// TIA Portal V16 export
// export: Created 2022-01-20T18:36:27.7444699Z, ExportSetting WithDefaults, DisplayName Totally Integrated Automation Portal, DisplayVersion V16, DisplayName TIA Portal Version Control Interface, DisplayVersion V16, DisplayName TIA Portal Openness, DisplayVersion V16, DisplayName STEP 7 Professional, DisplayVersion V16, DisplayName STEP 7 Safety, DisplayVersion V16, DisplayName WinCC Advanced, DisplayVersion V16
FUNCTION_BLOCK "TCPIP_COMMS"   // FB1, LAD
{ S7_Optimized_Access := 'TRUE' }
VERSION : 0.1
// stored: AutoNumber true, IsIECCheckEnabled false, IsRetainMemResEnabled false, MemoryReserve 100, SetENOAutomatically false, UDAEnableTagReadback false
   VAR
      TCON : Struct
         REQ : Bool;
         DONE : Bool;
         BUSY : Bool;
         ERROR : Bool;
         STATUS : UInt;
         DONESAVE : Bool;
      END_STRUCT;
      TDISCON : Struct
         REQ : Bool;
         DONE : Bool;
         BUSY : Bool;
         ERROR : Bool;
         DONESAVE : Bool;
         STATUS : UInt;
      END_STRUCT;
      TSEND : Struct
         REQ : Bool;
         DONE : Bool;
         BUSY : Bool;
         ERROR : Bool;
         DONESAVE : Bool;
         STATUS : UInt;
      END_STRUCT;
      TRCV : Struct
         EN_R : Bool;
         NDR : Bool;
         BUSY : Bool;
         ERROR : Bool;
         STATUS : UInt;
         RCVD_LEN : UDInt;
      END_STRUCT;
      ReceivedString : String;
      TCON_DB { ExternalAccessible := 'False'; ExternalVisible := 'False'; ExternalWritable := 'False'} : TCON;
      TDISCON_DB { ExternalAccessible := 'False'; ExternalVisible := 'False'; ExternalWritable := 'False'} : TDISCON;
      TSEND_DB { ExternalAccessible := 'False'; ExternalVisible := 'False'; ExternalWritable := 'False'} : TSEND;
      TRCV_DB { ExternalAccessible := 'False'; ExternalVisible := 'False'; ExternalWritable := 'False'} : TRCV;
   END_VAR
BEGIN

REGION Network 1: TCON
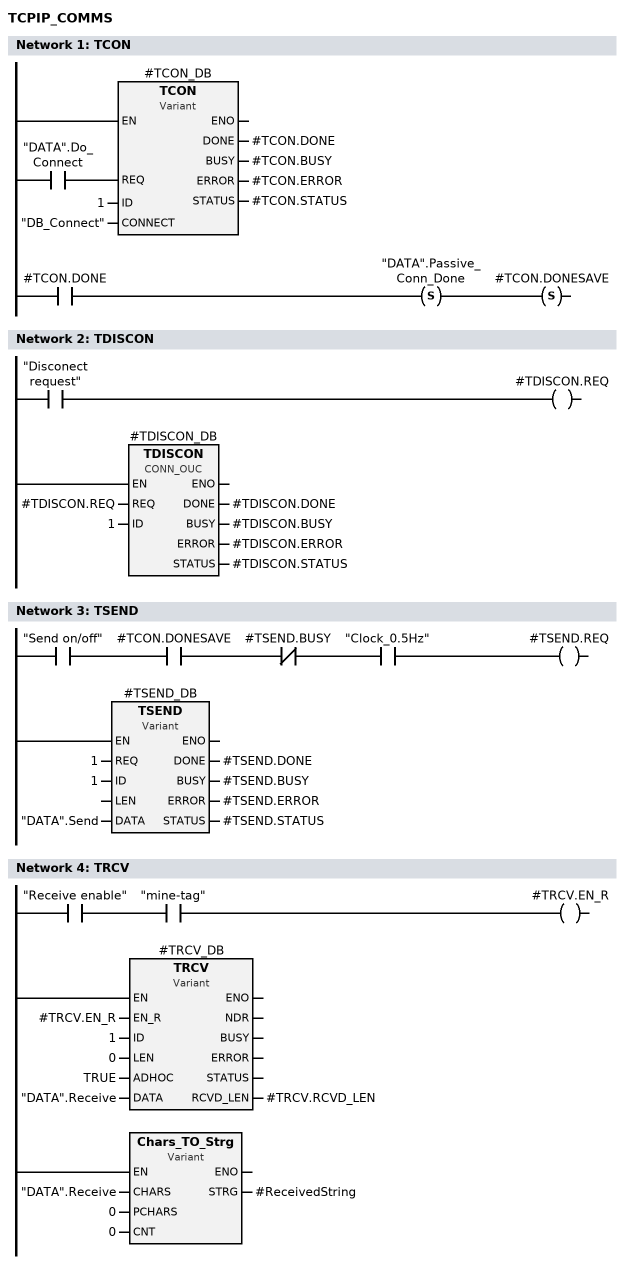
   RUNG wire#powerrail
      { S7_Templates := "[con_type := Variant, id_type := CONN_OUC]" } #TCON_DB.TCON(REQ := wire#w1, ID := 1, CONNECT := "DB_Connect", DONE => #TCON.DONE, BUSY => #TCON.BUSY, ERROR => #TCON.ERROR, STATUS => #TCON.STATUS)
   END_RUNG
   RUNG wire#powerrail
      Contact( "DATA".Do_Connect )
   END_RUNG wire#w1
   RUNG wire#powerrail
      Contact( #TCON.DONE )
      S_Coil( "DATA".Passive_Conn_Done )
      S_Coil( #TCON.DONESAVE )
   END_RUNG
   // the same network as SCL:
   #TCON_DB(REQ := "DATA".Do_Connect,   // TCON
            ID := 1,
            CONNECT := "DB_Connect",
            DONE => #TCON.DONE,
            BUSY => #TCON.BUSY,
            ERROR => #TCON.ERROR,
            STATUS => #TCON.STATUS);
   IF #TCON.DONE THEN
       "DATA".Passive_Conn_Done := TRUE;
       #TCON.DONESAVE := TRUE;
   END_IF;
END_REGION

REGION Network 2: TDISCON
   RUNG wire#powerrail
      Contact( "Disconect request" )
      Coil( #TDISCON.REQ )
   END_RUNG
   RUNG wire#powerrail
      { S7_Templates := "id_type := CONN_OUC" } #TDISCON_DB.TDISCON(REQ := #TDISCON.REQ, ID := 1, DONE => #TDISCON.DONE, BUSY => #TDISCON.BUSY, ERROR => #TDISCON.ERROR, STATUS => #TDISCON.STATUS)
   END_RUNG
   // the same network as SCL:
   #TDISCON.REQ := "Disconect request";
   #TDISCON_DB(REQ := #TDISCON.REQ,   // TDISCON
               ID := 1,
               DONE => #TDISCON.DONE,
               BUSY => #TDISCON.BUSY,
               ERROR => #TDISCON.ERROR,
               STATUS => #TDISCON.STATUS);
END_REGION

REGION Network 3: TSEND
   RUNG wire#powerrail
      Contact( "Send on/off" )
      Contact( #TCON.DONESAVE )
      I_Contact( #TSEND.BUSY )
      Contact( "Clock_0.5Hz" )
      Coil( #TSEND.REQ )
   END_RUNG
   RUNG wire#powerrail
      { S7_Templates := "[data_type := Variant, len_type := UDInt, id_type := CONN_OUC]" } #TSEND_DB.TSEND(REQ := 1, ID := 1, LEN :=, DATA := "DATA".Send, DONE => #TSEND.DONE, BUSY => #TSEND.BUSY, ERROR => #TSEND.ERROR, STATUS => #TSEND.STATUS)
   END_RUNG
   // the same network as SCL:
   #TSEND.REQ := "Send on/off" AND #TCON.DONESAVE AND NOT #TSEND.BUSY AND "Clock_0.5Hz";
   #TSEND_DB(REQ := 1,   // TSEND
             ID := 1,
             DATA := "DATA".Send,
             DONE => #TSEND.DONE,
             BUSY => #TSEND.BUSY,
             ERROR => #TSEND.ERROR,
             STATUS => #TSEND.STATUS);
END_REGION

REGION Network 4: TRCV
   RUNG wire#powerrail
      Contact( "Receive enable" )
      Contact( "mine-tag" )
      Coil( #TRCV.EN_R )
   END_RUNG
   RUNG wire#powerrail
      { S7_Templates := "[card := 1, ptr_type := Variant, value_type := UDInt, id_type := CONN_OUC]" } #TRCV_DB.TRCV(EN_R := #TRCV.EN_R, ID := 1, LEN := 0, ADHOC := TRUE, DATA := "DATA".Receive, NDR =>, BUSY =>, ERROR =>, STATUS =>, RCVD_LEN => #TRCV.RCVD_LEN)
   END_RUNG
   RUNG wire#powerrail
      { S7_Templates := "[ptr_type := Variant, str_type := String]" } Chars_TO_Strg(Chars := "DATA".Receive, pChars := 0, Cnt := 0, Strg => #ReceivedString)
   END_RUNG
   // the same network as SCL:
   #TRCV.EN_R := "Receive enable" AND "mine-tag";
   #TRCV_DB(EN_R := #TRCV.EN_R,   // TRCV
            ID := 1,
            LEN := 0,
            ADHOC := TRUE,
            DATA := "DATA".Receive,
            RCVD_LEN => #TRCV.RCVD_LEN);
   Chars_TO_Strg(Chars := "DATA".Receive, pChars := 0, Cnt := 0, Strg => #ReceivedString);
END_REGION
END_FUNCTION_BLOCK
